// TIA Portal V18 export
DATA_BLOCK "BoilerUnitStates"   // DB1
{ S7_Optimized_Access := 'TRUE' }
VERSION : 0.1
// stored: AutoNumber true, DBAccessibleFromOPCUA true, IsOnlyStoredInLoadMemory false, IsRetainMemResEnabled false, IsWriteProtectedInAS false, MemoryReserve 100
   VAR
      UnitStates { S7_SetPoint := 'True'} : "UDT_BoilerUnitState";
   END_VAR
BEGIN
END_DATA_BLOCK
